Staubli VAL3: getListTitle.pgx

public program getListTitle(string& x_sMsg (dimensions=1))
begin
  if save:nBoxType==1
    call language2:message(x_sMsg,1)
  elseIf save:nBoxType==2
    call language2:message(x_sMsg,2)
  endIf
end
